FUNCTION_BLOCK StateMachine
VAR_INPUT
END_VAR
VAR_OUTPUT
END_VAR
VAR
	InitDone: BOOL;
	NewState: POINTER TO State;
	CurrentState: POINTER TO State;
	DummyState: State;
	LastState: POINTER TO State := ADR(DummyState);
END_VAR

IF NOT InitDone THEN
	CurrentState := StartState();
ELSE
	CurrentState := CurrentState^.Transition();
END_IF

IF CurrentState <> LastState THEN
	LastState^.Stop();
	CurrentState^.Start();
	LastState := CurrentState;
END_IF

METHOD StartState : POINTER TO State
VAR_INPUT
END_VAR
END_METHOD

END_FUNCTION_BLOCK

(* stored: Version 1.1.0.1, ProductVersion 3.1.4024.3
   POU StateMachine: Id {394cde49-38b6-4844-a793-c5de2f4e2276}, SpecialFunc None
   Method StartState: Id {7f2e7588-16f9-4ffb-b547-ae26954dd9da} *)
